FUNCTION_BLOCK SAMPLE_BYTE (* Sample a single byte - see SAMPLE_1 *)
  (* Standard: 61499-1; Classification: Math; Function: Sampling; Type: BYTE *)
  (* Version 0.1, 2008-06-25, JHC, Holobloc Inc, Updated to new implementation. *)
  (* Version 0.0, 2006-05-28, JHC, Holobloc Inc *)
  (* Compiler header: package fb.rt.math; *)
  (* Compiler classdef: public class SAMPLE_BYTE extends ChangeSensor *)
  (* Compiler Java Sun JDK 1.6.0 *)
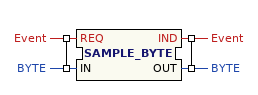
  EVENT_INPUT
    REQ WITH IN; (* Request to Sample *)
  END_EVENT
  EVENT_OUTPUT
    IND WITH OUT; (* Initial Sample or OUT changed *)
  END_EVENT
  VAR_INPUT
    IN : BYTE; (* Data to Sample *)
  END_VAR
  VAR_OUTPUT
    OUT : BYTE; (* Sampled Data *)
  END_VAR
END_FUNCTION_BLOCK
